VISUALIZATION VISU_MTCSSystemBackground  // 2x2
END_VISUALIZATION

(* stored: Version 1.1.0.1, ProductVersion 3.1.0.36
   Visu VISU_MTCSSystemBackground: Id {56631fcc-563c-4d32-96d6-8d65c24f1b4a} *)
